FUNCTION IsBetween : BOOL
VAR_INPUT
	value: 	LREAL;
	minV:	LREAL;
	maxV:	LREAL;
END_VAR
VAR
END_VAR

IsBetween := value > minV AND value < maxV;

END_FUNCTION

(* stored: Version 1.1.0.1, ProductVersion 3.1.4026.8
   POU IsBetween: Id {30980012-edae-416d-9aac-47ae41f64e5a}, SpecialFunc None *)
